INTERFACE I_RpcHeaderAccessor

PROPERTY PUBLIC ContentType_Json : T_MAXSTRING
GET
END_GET
END_PROPERTY

METHOD PUBLIC TryGetAcceptResponseFormatFromRequest : BOOL
VAR_INPUT
	Request : I_Request;
	Destination : ANY;
END_VAR
END_METHOD

METHOD PUBLIC TryGetContentTypeFromRequest : BOOL
VAR_INPUT
	Request : I_Request;
	Destination : ANY;
END_VAR
END_METHOD

METHOD PUBLIC TryGetMethodNameFromRequest : BOOL
VAR_INPUT
	Request : I_Request;
	Destination : ANY;
END_VAR
END_METHOD

METHOD PUBLIC TryGetTypeFromRequest : BOOL
VAR_INPUT
	Request : I_Request;
	Destination : ANY;
END_VAR
END_METHOD

END_INTERFACE

(* stored: Version 1.1.0.1, ProductVersion 3.1.4026.13
   Itf I_RpcHeaderAccessor: Id {f35e86d1-9544-423b-baa9-95563a212d8e}
   Property ContentType_Json: Id {68e0d632-0fa2-48f7-a1ce-4c0f0ca94bee}
   Get Get: Id {c6f6f016-d44a-4fac-87d5-261a6242aa17}
   Method TryGetAcceptResponseFormatFromRequest: Id {44e47596-14af-435c-a905-1b33e3933d11}
   Method TryGetContentTypeFromRequest: Id {b823ff68-23cc-4391-a4d1-c6ea637a6da1}
   Method TryGetMethodNameFromRequest: Id {3b61b50d-08b9-43e1-8264-6cb5ee2de134}
   Method TryGetTypeFromRequest: Id {2d5d29cd-3819-43cd-8290-84fbd5f32847} *)
